FUNCTION TryConvert_TIME_TO_DATE : BOOL
VAR_INPUT
	in : TIME;
	out : REFERENCE TO DATE;
END_VAR

out := TIME_TO_DATE(in);
TryConvert_TIME_TO_DATE := TRUE;

END_FUNCTION

(* stored: Version 1.1.0.1, ProductVersion 3.1.4024.12
   POU TryConvert_TIME_TO_DATE: Id {02b803d0-3324-4a14-a4c9-0dc224407b1d}, SpecialFunc None *)
